// Monitors the Amphos MRC input signal for errors
FUNCTION_BLOCK FB_AmphosMRC
VAR_INPUT
    bAmphosOn : BOOL; // Whether the Amphos is turned on
    bMRC : BOOL; // Error signal. Signal should normally be high
END_VAR
VAR_OUTPUT
    {attribute 'pytmc' := '
        pv: ERROR
        io: i
        field: OSV MAJOR
        field: ZSV NO_ALARM
        field: ZNAM OK
        field: ONAM ERROR
    '}
    bError : BOOL; // Whether an error was detected. Error should go back to normal on its own
END_VAR
VAR
END_VAR

(* Set error flag if amphos is on and the MRC has an error *)
bError := bAmphosOn AND NOT bMRC;

END_FUNCTION_BLOCK

(* stored: Version 1.1.0.1, ProductVersion 3.1.4024.6
   POU FB_AmphosMRC: Id {47914c31-5a87-4cd7-bcb9-0928e1947083}, SpecialFunc None *)
